(* IEC 61131-3 sources: programs/VI-54/VI-54_20171205/VI-54_20171205/Stations/PLC_VI54/VI-54_171014/Class/MainRecipe, 1 file *)

(* ---- MainRecipe.st ---- *)
(*!
<Class
	Name               = "MainRecipe"
	Revision           = "0.0"
	RealtimeTask       = "false"
	CyclicTask         = "false"
	BackgroundTask     = "false"
	Sigmatek           = "false"
	OSInterface        = "false"
	HighPriority       = "false"
	Automatic          = "false"
	UpdateMode         = "Prescan"
	SharedCommandTable = "true"
	Objectsize         = "(630,120)">
	<Channels>
		<Server Name="ClassSvr" Visualized="false" Initialize="false" WriteProtected="true" Retentive="false"/>
		<Client Name="DataRecipe" Required="true" Internal="true"/>
	</Channels>
	<Network Name="MainRecipe">
		<!-- List of Components in this network -->
		<Components>
			<Object
				Name       = "DataRecipe"
				Class      = "MerkerEx"
				Position   = "(210,180)"
				Visualized = "true"
				Remotely   = "true">
				<Channels>
					<Server Name="m_udLength"/>
					<Client Name="ThreadSafe" Value="0"/>
				</Channels>
			</Object>
		</Components>
		<Comments>
		</Comments>
		<!-- List of Connections in this network -->
		<Connections>
			<Connection Source="this.DataRecipe" Destination="DataRecipe.m_udLength"/>
		</Connections>
		<!-- Headerfiles -->
		<Options>
		</Options>
	</Network>
</Class>
*)
MainRecipe : CLASS
  //Servers:
	ClassSvr 	: SvrChCmd_DINT;
  //Clients:
	DataRecipe 	: CltChCmd_MerkerEx;
  //Variables:
		RecipePtr 	: ^DataRecipeStr;
		MyFirstScan 	: DINT;
  //Functions:

	FUNCTION VIRTUAL GLOBAL Init;

	FUNCTION GLOBAL GetPointer
		VAR_OUTPUT
			Ptr 	: ^DataRecipeStr;
		END_VAR;
  //Tables:
	FUNCTION @STD
		VAR_OUTPUT
			ret_code	: CONFSTATES;
		END_VAR;
	FUNCTION GLOBAL TAB @CT_;
END_CLASS;

#pragma using MerkerEx

FUNCTION VIRTUAL GLOBAL MainRecipe::Init

  // Check size
  if DataRecipe.GetSize() <> sizeof(DataRecipeStr) then
    DataRecipe.SetSize(udSize:= sizeof(DataRecipeStr));
  end_if;

  // Set pointer
  if MyFirstScan = 0 then
    RecipePtr$^USINT := DataRecipe.GetDataPtr();
    MyFirstScan := 1;
  end_if;

END_FUNCTION

FUNCTION GLOBAL MainRecipe::GetPointer
	VAR_OUTPUT
		Ptr 	: ^DataRecipeStr;
	END_VAR

  Ptr := RecipePtr;

END_FUNCTION
